# EPICS substitutions: iocs/photronIOC/iocBoot/iocPhotron/templates/photronExtIO.substitutions
file "$(ADPHOTRON)/photronApp/Db/PhotronExtIOPort.db"
{
pattern
{P,		R,		N,	PORT,	ADDR,	TIMEOUT}
{pho:,	cam1:,	1,	PHO1,	0,		1}
{pho:,	cam1:,	2,	PHO1,	0,		1}
{pho:,	cam1:,	3,	PHO1,	0,		1}
{pho:,	cam1:,	4,	PHO1,	0,		1}
}
